// Some aggregate that has implemented a process for demonstration.
FUNCTION_BLOCK FB_ProcAggregateB EXTENDS FB_BA_AggregateB
VAR
	Delay			: TON					:= (PT:=T#7S);
	Process			: FB_BA_Process			:= (iParent:=THIS^);
END_VAR

SUPER^();

Delay(IN := (bActiveEn AND bActiveVal));
Process(
	bEn := Delay.IN,
	bVal := (NOT Delay.Q)
);

END_FUNCTION_BLOCK

(* stored: Version 1.1.0.1, ProductVersion 3.1.4024.9
   POU FB_ProcAggregateB: Id {e7e2e93b-b12f-4626-a312-91fafef05993}, SpecialFunc None *)
